(* IEC 61131-3 sources: ICSQuartz/benchmarks/oscat_basic_findp/src, 1 file *)

(* ---- program.st ---- *)
PROGRAM PLC_PRG
VAR_INPUT
    in_pos: INT;
    in_str: STRING;
    in_src: STRING;
END_VAR

FINDP(in_str, in_src, in_pos);

END_PROGRAM
